TYPE DUT_HMI_15 :
STRUCT
	Manuals : DUT_HMI_15_MANUALS;
	ProductStatus 	: eProductStatus;
	State			: eStationState;
	EVDiagnostic 	: ARRAY[0..20] OF DUT_HMI_EV_Diagnostic;
	EVInfo			: ARRAY[0..CNC.NUM_MAX_MANUALS_15-1] OF DUT_HMI_EV_Info;
	Status			: USINT;
	CycleTime		: STRING;
END_STRUCT
END_TYPE

(* stored: Version 1.1.0.1, ProductVersion 3.1.4024.15
   DUT DUT_HMI_15: Id {9819a0e9-49c1-4202-a156-ff8f859ed66b} *)
